# EPICS StreamDevice protocol: Lakeshore_460Sup/devLakeshore_460.proto
Terminator = '\r\n';
ReplyTimeout = 2000;
ReadTimeout = 2000;
WriteTimeout = 2000;

getIDN {
    out "*IDN?";
	wait 50;
    #Read no more that 39 chars (EPICS limit)
    in "LSCI,MODEL460,0,%s";
    ExtraInput = Ignore;
}

# Channel arguments passed though as \$1 ##

getMagneticFieldReading
{
	out "CHNL \$1;FIELD?";
	wait 50;
	in "%*{+|-}%f";
	@mismatch { in 5; }
	ExtraInput = Ignore;
}

getMagneticFieldUnitsMultiplier
{
	out "CHNL \$1;FIELDM?";
	in "%s"
}

getMagneticFieldUnits
{
    out "UNIT?";
	wait 50;
    in "%s";
}

setMagneticFieldUnits
{
    out "UNIT %{G|T}";
	wait 50;
	@init { out "UNIT?"; in "%s"; wait 50; }
}

getStatus
{
    out "CHNL \$1;ONOFF?";
    in "%d";
	wait 50;
}

setStatus
{
	out "CHNL \$1;ONOFF %{0|1}";
	wait 50;
	@init { out "CHNL \$1;ONOFF?"; in "%d"; wait 50; }
}

getACDCFieldReading {
	out "CHNL \$1;ACDC?";
	wait 50;
	in "%d";
}

setACDCFieldReading {
	out "CHNL \$1;ACDC %{0|1}";
	wait 50;
	@init { out "CHNL \$1;ACDC??"; in "%d"; wait 50; }
}

getPRMSReading {
	out "CHNL \$1;PRMS?";
	wait 50;
	in "%d";
}

setPRMSReading {
	out "CHNL \$1;PRMS %{0|1}";
	wait 50;
}

getFilter {
	out "CHNL \$1;FILT?";
	wait 50;
	in "%d";
}

setFilter {
	out "CHNL \$1;FILT %{0|1}";
	wait 50;
}

getRelMode {
	out "CHNL \$1;REL?";
	wait 50;
	in "%d";
}

setRelMode {
	out "CHNL \$1;REL %{0|1}";
	wait 50;
}

getMaxHold {
	out "CHNL \$1;MAX?";
	wait 50;
	in "%d";
}

setMaxHold {
	out "CHNL \$1;MAX %{0|1}";
	wait 50;
}

getAutoRange {
	out "CHNL \$1;AUTO?";
	wait 50;
	in "%d";
}

setAutoRange {
	out "CHNL \$1;AUTO %{0|1}";
	wait 50;
}

getAllFields {
	out "ALLF?";
	wait 50;
	in "%f";
}

getSource {
	out "VSRC?";
	wait 50;
	in "%d";
}

setSource {
	out "VSRC %d";
	wait 50;
}

getChannel {
	out "CHNL?";
	wait 50;
	in "%s";
}

setChannel {
	out "CHNL %d";
	wait 50;
}

getFWin {
	out "CHNL \$1;FWIN?";
	wait 50;
	in "%d";
}

setFWin {
	out "CHNL \$1;FWIN %d";
	wait 50;
}

getFNum {
	out "CHNL \$1;FNUM?";
	wait 50;
	in "%d";
}

setFNum {
	out "CHNL \$1;FNUM %d";
	wait 50;
}

getManualRange {
	out "CHNL \$1;RANGE?";
	in "%d";
}

setManualRange {
	out "CHNL \$1;RANGE %d";
}

getMaxReading {
	out "CHNL \$1;MAXR?";
	in "%f";
	ExtraInput = Ignore;
}

getRelModeReading {
	out "CHNL \$1;RELR?";
	in "%f";
	ExtraInput = Ignore;
}
